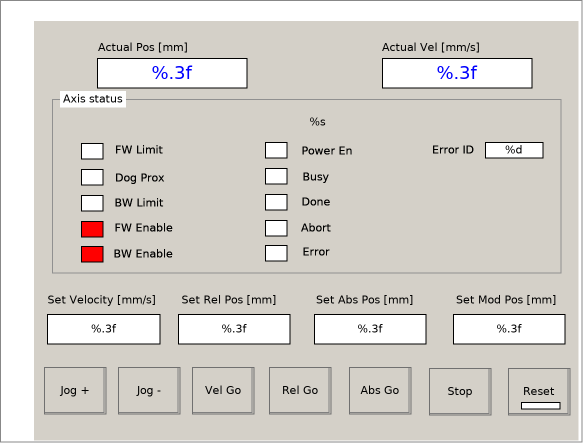
VISUALIZATION Axis_Page  // 583x443
VAR_IN_OUT
	userdata : Axis_HMI_Struct;
END_VAR
    Rectangle (33,20 546x421)
    Button (44,367 62x47), "Jog +"
        tap userdata.bJog_F
    GroupBox (52,91 509x182), "Axis status"
        Rectangle (29,52 22x16), colour toggle: userdata.bFW_LimitSwith
        Rectangle (29,104 22x16), colour toggle: userdata.bBW_LimitSwith
        Rectangle (29,78 22x16), colour toggle: userdata.bDog_PointSwith
        Rectangle (29,130 22x16), colour toggle: userdata.bForwordEnable
        Rectangle (29,155 22x16), colour toggle: userdata.bBackwordEnable
        Rectangle (213,51 22x16), colour toggle: userdata.bPowerEn
        Rectangle (213,103 22x16), colour toggle: userdata.bDone
        Rectangle (213,77 22x16), colour toggle: userdata.bBusy
        Rectangle (213,129 22x16), colour toggle: userdata.bAborted
        Rectangle (213,154 22x16), colour toggle: userdata.bError
        Rectangle (433,51 58x16), "%d", text variable: userdata.nErrorID, colour toggle: userdata.nErrorID
        Rectangle (113,21 305x20), "%s", text variable: userdata.cErrorTXT
        Label (12,44 150x30), "FW Limit"
        Label (12,97 150x30), "BW Limit"
        Label (17,122 150x30), "FW Enable"
        Label (17,148 149x30), "BW Enable"
        Label (13,72 150x30), "Dog Prox"
        Label (200,45 150x30), "Power En"
        Label (189,71 150x30), "Busy"
        Label (189,122 150x30), "Abort"
        Label (189,96 150x30), "Done"
        Label (189,146 150x30), "Error"
        Label (326,44 150x30), "Error ID"
    Rectangle (81,143 22x16), colour toggle: userdata.bFW_LimitSwith
    Rectangle (81,195 22x16), colour toggle: userdata.bBW_LimitSwith
    Rectangle (81,169 22x16), colour toggle: userdata.bDog_PointSwith
    Rectangle (81,221 22x16), colour toggle: userdata.bForwordEnable
    Rectangle (81,246 22x16), colour toggle: userdata.bBackwordEnable
    Rectangle (265,142 22x16), colour toggle: userdata.bPowerEn
    Rectangle (265,194 22x16), colour toggle: userdata.bDone
    Rectangle (265,168 22x16), colour toggle: userdata.bBusy
    Rectangle (265,220 22x16), colour toggle: userdata.bAborted
    Rectangle (265,245 22x16), colour toggle: userdata.bError
    Rectangle (485,142 58x16), "%d", text variable: userdata.nErrorID, colour toggle: userdata.nErrorID
    Rectangle (165,112 305x20), "%s", text variable: userdata.cErrorTXT
    Label (64,135 150x30), "FW Limit"
    Label (64,188 150x30), "BW Limit"
    Label (69,213 150x30), "FW Enable"
    Label (69,239 149x30), "BW Enable"
    Label (65,163 150x30), "Dog Prox"
    Label (252,136 150x30), "Power En"
    Label (241,162 150x30), "Busy"
    Label (241,213 150x30), "Abort"
    Label (241,187 150x30), "Done"
    Label (241,237 150x30), "Error"
    Label (378,135 150x30), "Error ID"
    Rectangle (97,58 150x30), "%.3f", text variable: userdata.Axis_ref.NcToPlc.ActPos
    Rectangle (382,58 150x30), "%.3f", text variable: userdata.Axis_ref.NcToPlc.ActVelo
    Rectangle (47,314 113x30), "%.3f", text variable: userdata.fSetVel_Man
        OnMouseDown: write the text variable via Edit
    Button (118,367 62x47), "Jog -"
        tap userdata.bJog_B
    Button (192,367 62x47), "Vel Go"
        tap userdata.bVelGo_Man
    Button (349,367 62x47), "Abs Go"
        tap userdata.bAbsGo_Man
    Button (269,367 62x47), "Rel Go"
        tap userdata.bRelGo_Man
    Button (429,368 62x47), "Stop"
        tap userdata.bStop_Man
    Button (508,368 62x47), "Reset"
        tap userdata.bReset_Man
    Label (69,37 148x21), "Actual Pos [mm]"
    Label (357,37 148x21), "Actual Vel [mm/s]"
    Label (31,285 138x30), "Set Velocity [mm/s]"
    Rectangle (178,314 112x30), "%.3f", text variable: userdata.fSetRelPos_Man
        OnMouseDown: write the text variable via Edit
    Rectangle (314,314 112x30), "%.3f", text variable: userdata.fSetAbsPos_Man
        OnMouseDown: write the text variable via Edit
    Label (154,285 150x30), "Set Rel Pos [mm]"
    Label (290,285 150x30), "Set Abs Pos [mm]"
    Rectangle (453,314 112x30), "%.3f", text variable: userdata.fSetModPos_Man
        OnMouseDown: write the text variable via Edit
    Label (432,285 149x30), "Set Mod Pos [mm]"
    RoundedRectangle (521,402 39x7), colour toggle: userdata.bError
END_VISUALIZATION

(* stored: Version 1.1.0.1, ProductVersion 3.1.4018.5
   Visu Axis_Page: Id {dcb4bcaf-ea04-4509-a713-c953a54a954b} *)
